// TIA Portal V18 export
DATA_BLOCK "DB 335"   // DB335
{ S7_Optimized_Access := 'FALSE' }
AUTHOR : AWP_S7P
FAMILY : WEB
VERSION : 0.1
   VAR
      MAGIC : DWord := DW#16#4157_5046;
      CONSISTENCY_TAG : DWord := 252882973;
